// TIA Portal V20 export
VAR_GLOBAL   // PLC tag table "LNK_Const_Gen"
END_VAR
VAR_GLOBAL CONSTANT   // user constants
   LNK_MAGIC : Word := 16#4753;   // FRAME header magic 'GS' / FRAME 헤더 매직 'GS'
   LNK_VERSION : USInt := 1;   // FRAME header version / FRAME 헤더 버전
   LNK_FMT_JSON : USInt := 1;   // Payload format JSON / 페이로드 포맷 JSON
   LNK_FMT_BIN : USInt := 2;   // Payload format BIN (Serialize) / 페이로드 포맷 BIN (Serialize)
   LNK_HDR_LEN : DInt := 16;   // FRAME header length (bytes) / FRAME 헤더 길이 (B)
   LNK_MAX_PAYLOAD : DInt := 8176;   // PLC receive payload / line max (bytes) / PLC 수신 페이로드 / 줄 최대 (B)
   LNK_MSG_HELLO : UInt := 1;   // Message id Hello (LNK_Hello) / 메시지 ID Hello
   LNK_MSG_HEARTBEAT : UInt := 2;   // Message id Heartbeat (no payload) / 메시지 ID Heartbeat (페이로드 없음)
   LNK_MSG_ACK : UInt := 30;   // Message id Ack (LNK_Ack) / 메시지 ID Ack
   LNK_MSG_FIXTURE : UInt := 40;   // Message id Fixture (LNK_Fixture) / 메시지 ID Fixture
   LNK_MSG_FIXTURECMD : UInt := 41;   // Message id FixtureCmd (LNK_FixtureSub) / 메시지 ID FixtureCmd
   LNK_MSG_JSONONLY : UInt := 42;   // Message id JsonOnly (LNK_FixtureSub) / 메시지 ID JsonOnly
   LNK_MSG_MISSING : UInt := 50;   // Message id Missing (LNK_DoesNotExist) / 메시지 ID Missing
   LNK_SIG_HELLO : DWord := 16#BFAD9982;   // UDT signature LNK_Hello / UDT 시그니처 LNK_Hello
   LNK_SIG_ACK : DWord := 16#FF5482FF;   // UDT signature LNK_Ack / UDT 시그니처 LNK_Ack
   LNK_SIG_FIXTURE : DWord := 16#EB2E5DE0;   // UDT signature LNK_Fixture / UDT 시그니처 LNK_Fixture
   LNK_SIG_FIXTURECMD : DWord := 16#AFBB75A6;   // UDT signature LNK_FixtureSub / UDT 시그니처 LNK_FixtureSub
   LNK_SIG_JSONONLY : DWord := 16#AFBB75A6;   // UDT signature LNK_FixtureSub / UDT 시그니처 LNK_FixtureSub
   LNK_LEN_HELLO : DInt := 28;   // Serialized size LNK_Hello (bytes) / 직렬화 크기 LNK_Hello (B)
   LNK_LEN_ACK : DInt := 48;   // Serialized size LNK_Ack (bytes) / 직렬화 크기 LNK_Ack (B)
   LNK_LEN_FIXTURE : DInt := 170;   // Serialized size LNK_Fixture (bytes) / 직렬화 크기 LNK_Fixture (B)
   LNK_LEN_FIXTURECMD : DInt := 26;   // Serialized size LNK_FixtureSub (bytes) / 직렬화 크기 LNK_FixtureSub (B)
   LNK_LEN_JSONONLY : DInt := 26;   // Serialized size LNK_FixtureSub (bytes) / 직렬화 크기 LNK_FixtureSub (B)
   LNK_JMAX_HELLO : DInt := 236;   // Max JSON envelope length Hello (bytes) / JSON 엔벨로프 최대 길이 Hello (B)
   LNK_JMAX_ACK : DInt := 347;   // Max JSON envelope length Ack (bytes) / JSON 엔벨로프 최대 길이 Ack (B)
   LNK_JMAX_FIXTURE : DInt := 999;   // Max JSON envelope length Fixture (bytes) / JSON 엔벨로프 최대 길이 Fixture (B)
   LNK_JMAX_FIXTURECMD : DInt := 187;   // Max JSON envelope length FixtureCmd (bytes) / JSON 엔벨로프 최대 길이 FixtureCmd (B)
   LNK_JMAX_JSONONLY : DInt := 185;   // Max JSON envelope length JsonOnly (bytes) / JSON 엔벨로프 최대 길이 JsonOnly (B)
   LNK_REGISTRY_HASH : DWord := 16#C3CAA074;   // Message registry hash (crc32, wire-spec 5) / 메시지 레지스트리 해시 (crc32)
   LNK_ERR_OK : Int := 0;   // Link error: OK / 링크 오류: 정상
   LNK_ERR_BAD_MAGIC : Int := 1;   // Link error: bad FRAME magic / 링크 오류: FRAME 매직 불일치
   LNK_ERR_BAD_VERSION : Int := 2;   // Link error: bad FRAME version / 링크 오류: FRAME 버전 불일치
   LNK_ERR_UNKNOWN_TYPE : Int := 3;   // Link error: unknown message type / 링크 오류: 알 수 없는 메시지
   LNK_ERR_SIG_MISMATCH : Int := 4;   // Link error: BIN layout signature mismatch / 링크 오류: BIN 시그니처 불일치
   LNK_ERR_BAD_LENGTH : Int := 5;   // Link error: bad length / 링크 오류: 길이 오류
   LNK_ERR_PARSE : Int := 6;   // Link error: parse error / 링크 오류: 파싱 오류
   LNK_ERR_FORMAT_NOT_ALLOWED : Int := 7;   // Link error: format not allowed (BIN over NDJSON) / 링크 오류: 허용되지 않는 포맷 (NDJSON 위 BIN)
   LNK_ERR_DIR_NOT_ALLOWED : Int := 8;   // Link error: direction not allowed / 링크 오류: 허용되지 않는 방향
   LNK_ERR_BUSY : Int := 9;   // Link error: busy / 링크 오류: 처리 중
   LNK_ERR_NO_PENDING : Int := 10;   // Link error: nothing pending / 링크 오류: 대기 항목 없음
END_VAR
